FUNCTION_BLOCK ABSTRACT fbComponent IMPLEMENTS ITaskContainer
VAR	
	{attribute addProperty Name "Components' message"}
	{attribute clr [ReadOnly()]}
	_message : STRING(255);
	{attribute 'hide'}
	_lock : INT;		
END_VAR

METHOD PROTECTED Info
VAR_INPUT
	inMessage : STRING(255);
END_VAR
_message := inMessage;
END_METHOD

PROPERTY Lock : INT
GET
Lock := _lock;
END_GET
SET
_lock := Lock;
END_SET
END_PROPERTY

METHOD PUBLIC Manual
THIS^.ManualControl();
END_METHOD

METHOD PROTECTED ABSTRACT ManualControl
END_METHOD

END_FUNCTION_BLOCK

(* stored: Version 1.1.0.1, ProductVersion 3.1.4024.5
   POU fbComponent: Id {3a3f5739-2f9b-4ddf-a7b9-4efe8f16c6da}, SpecialFunc None
   Method Info: Id {4f2a9d49-7508-43d1-b8ca-30b80e325488}
   Property Lock: Id {894ca00a-deca-4836-9aec-96c7e557d980}
   Get Get: Id {d89713ca-8085-4f32-87d3-2686281caaa1}
   Set Set: Id {706a0668-cc90-458b-a90d-1300a332f7f5}
   Method Manual: Id {ebaeaa1d-acc8-400b-b205-2722550bd13c}
   Method ManualControl: Id {06f21b03-8098-4a97-9d0b-2e50bc362267} *)
